TYPE T_Ctrl_SIf_PBC_Ilk :
STRUCT
END_STRUCT
END_TYPE

(* stored: Version 1.1.0.1, ProductVersion 3.1.0.36
   DUT T_Ctrl_SIf_PBC_Ilk: Id {dd909d94-86bd-464c-9a57-68ed8bd899bf} *)
